TYPE ST_TCLevel :
STRUCT
	
		stGblParam: ST_TCSeqParam;
		fbTCLevelSeq: FB_TCLevelSeq;
		
END_STRUCT
END_TYPE

(* stored: Version 1.1.0.1, ProductVersion 3.1.4022.10
   DUT ST_TCLevel: Id {a0032924-8f7f-43a6-af76-be93511dca3e} *)
